{attribute 'GeneratedUsingTerminal: EK1100-0000-0018'}
{attribute addProperty BoxType "EK1100-0000-0018"}
{attribute addProperty Id "Beckhoff_EP3xxxEK1122Beckhoff_EP3xxxEK1122_7B33BCBC3196"}
{attribute addProperty CRC "88620096"}
{attribute addProperty Size "3196"}
{attribute addProperty Name "Beckhoff EP3xxx"}
TYPE Beckhoff_EP3xxx_05483C40 EXTENDS EK1100_1FC0878B :
STRUCT
	{attribute addProperty Name "Beckhoff EP3xxxEK1122"}
	{attribute addProperty PreviousPort "Beckhoff EP3xxx : B"}
	Beckhoff_EP3xxxEK1122 : Beckhoff_EP3xxxEK1122_7B33BCBC;
END_STRUCT
END_TYPE

(* stored: Version 1.2.0.0, ProductVersion 3.1.4024.11
   DUT Beckhoff_EP3xxx_05483C40: Id {d5ae0b09-513a-46e0-bdbc-675d7565e34c} *)
